// TIA Portal V20 export
VAR_GLOBAL   // PLC tag table "Unit1Em5"
   "BA010AZCRPM04.06" AT %Q2012.6 : Bool;   // NG & MANUAL INPUT CYLINDER DOWN
   "BA010AZCRPM04.07" AT %Q2012.7 : Bool;   // NG & MANUAL INPUT CYLINDER UP
   "BA010AZCRPM04.10" AT %Q2013.0 : Bool;   // MAGAZINE LOCK CYLINDER UP
   "BA010AZCRPM04.11" AT %Q2013.1 : Bool;   // MAGAZINE LOCK CYLINDER DOWN
   "BA010AZCRBK06.00" AT %I1020.0 : Bool;   // NG & MANUAL INPUT CYLINDER UP
   "BA010AZCRBK06.01" AT %I1020.1 : Bool;   // MAGAZINE LOCK CYLINDER DOWN
   "BA010AZCRBK06.02" AT %I1020.2 : Bool;   // NG & MANUAL INPUT PAD VACUUM PRESSURE SWITCH
   "BA010AZCRBK06.07" AT %I1020.7 : Bool;   // NG & MANUAL INPUT MAGAZINE ELECTRODE DETECTION SENSOR
   "BA010AZCRBK06.10" AT %I1021.0 : Bool;   // NG & MANUAL INPUT CYLINDER DOWN
   "BA010AZCRBK06.11" AT %I1021.1 : Bool;   // MAGAZINE LOCK CYLINDER UP
   "BA010AZCRBK06.12" AT %I1021.2 : Bool;   // NG & MANUAL INPUT VIBRATOR VACUUM PRESSURE SWITCH
   "BA010AZCRBK06.14" AT %I1021.4 : Bool;   // NG & MANUAL INPUT ELECTRODE DETECTION SENSOR
   "BA010AZCRBK06.17" AT %I1021.7 : Bool;   // NG & MANUAL INPUT MAGAZINE DETECTION SENSOR
   "BA010AZCRBK07.06" AT %I1024.6 : Bool;   // NG & MANUAL INPUT MAGAZINE FULL SENSOR
   "BA010AZCRBK09.02" AT %Q2104.2 : Bool;   // NG & MANUAL INPUT PAD VACUUM ON
   "BA010AZCRBK09.03" AT %Q2104.3 : Bool;   // NG & MANUAL INPUT PAD VACUUM OFF
   "BA010AZCRBK09.04" AT %Q2104.4 : Bool;   // NG & MANUAL INPUT VIBRATOR VACUUM ON
   "BA010AZCRBK09.05" AT %Q2104.5 : Bool;   // NG & MANUAL INPUT VIBRATOR VACUUM OFF
   "BA010AZCRBK09.00" AT %Q2104.0 : Bool;   // NG & MANUAL INPUT VIBRATOR-1 ON
   "BA010AZCRBK09.01" AT %Q2104.1 : Bool;   // NG & MANUAL INPUT VIBRATOR-1 OFF
   "BA010AZCRBK09.06" AT %Q2104.6 : Bool;   // NG & MANUAL INPUT VIBRATOR-2 ON
   "BA010AZCRBK09.07" AT %Q2104.7 : Bool;   // NG & MANUAL INPUT VIBRATOR-2 OFF
   "BA010AZCRBK07.07" AT %I1024.7 : Bool;   // MAGAZINE Z-AXIS SAFETY PIN POSITION SENSOR
END_VAR
VAR_GLOBAL CONSTANT   // user constants
   U1EM5_NO_OF_AXES : USInt := 2;   // Starts with 1. E.g., the value 4 means that 4 axes exist.
   DR7_RatedTorque : LReal := 1.27;   // NgManualInputAxisY
   DR8_RatedTorque : LReal := 0.41;   // MagazineAxisZ
   U1EM5_JOB01 : DInt := 1;
   U1EM5_JOB02 : DInt := 2;
   U1EM5_JOB03 : DInt := 3;
   U1EM5_JOB04 : DInt := 4;
   U1EM5_JOB05 : DInt := 5;
   U1EM5_JOB06 : DInt := 6;
   U1EM5_JOB07 : DInt := 7;
   U1EM5_JOB08 : DInt := 8;
   U1EM5_JOB09 : DInt := 9;
   U1EM5_JOB10 : DInt := 10;
   U1EM5_JOB11 : DInt := 11;
   U1EM5_JOB12 : DInt := 12;
   U1EM5_JOB13 : DInt := 13;
   U1EM5_JOB14 : DInt := 14;
   U1EM5_JOB15 : DInt := 15;
   U1EM5_JOB16 : DInt := 16;
   U1EM5_JOB17 : DInt := 17;
   U1EM5_JOB18 : DInt := 18;
   U1EM5_JOB19 : DInt := 19;
   U1EM5_JOB20 : DInt := 20;
   U1EM5_JOB21 : DInt := 21;
   U1EM5_JOB22 : DInt := 22;
   U1EM5_JOB23 : DInt := 23;
   U1EM5_JOB24 : DInt := 24;
   U1EM5_JOB25 : DInt := 25;
   U1EM5_JOB26 : DInt := 26;
   U1EM5_JOB27 : DInt := 27;
   U1EM5_JOB28 : DInt := 28;
   U1EM5_JOB29 : DInt := 29;
   U1EM5_JOB30 : DInt := 30;
   U1EM5_JOB31 : DInt := 31;
   U1EM5_JOB32 : DInt := 32;
   U1EM5_JOB33 : DInt := 33;
   U1EM5_JOB34 : DInt := 34;
   U1EM5_JOB35 : DInt := 35;
   U1EM5_JOB36 : DInt := 36;
   U1EM5_JOB37 : DInt := 37;
   U1EM5_JOB38 : DInt := 38;
   U1EM5_JOB39 : DInt := 39;
   U1EM5_JOB40 : DInt := 40;
   U1EM5_JOB41 : DInt := 41;
   U1EM5_JOB42 : DInt := 42;
   U1EM5_JOB43 : DInt := 43;
   U1EM5_JOB44 : DInt := 44;
   U1EM5_JOB45 : DInt := 45;
   U1EM5_JOB46 : DInt := 46;
   U1EM5_JOB47 : DInt := 47;
   U1EM5_JOB48 : DInt := 48;
   U1EM5_JOB49 : DInt := 49;
   U1EM5_JOB50 : DInt := 50;
END_VAR
